FUNCTION_BLOCK ConvertToForce (* Basic Function Block Type *)
  (* Standard: 61499-2 *)
  (* Version 0.0, 8/12/2014, valvya, nxtControl GmbH, Template *)
  PACKAGE Main;
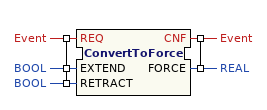
  EVENT_INPUT
    REQ WITH EXTEND, RETRACT; (* Normal Execution Request *)
  END_EVENT
  EVENT_OUTPUT
    CNF WITH FORCE; (* Execution Confirmation *)
  END_EVENT
  VAR_INPUT
    EXTEND : BOOL; (* Input event qualifier *)
    RETRACT : BOOL;
  END_VAR
  VAR_OUTPUT
    FORCE : REAL; (* Output event qualifier *)
  END_VAR
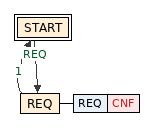
  EC_STATES
    START; (* Initial State *)
    REQ : REQ -> CNF; (* Normal execution *)
  END_STATES
  EC_TRANSITIONS
    START TO REQ := REQ;
    REQ TO START := 1;
  END_TRANSITIONS
  ALGORITHM REQ IN ST: (* Normally executed algorithm *)
IF EXTEND THEN FORCE:=100;
  ELSIF RETRACT THEN FORCE:=-100;
  ELSE  FORCE :=0;
END_IF;
  END_ALGORITHM
END_FUNCTION_BLOCK
